Universal Robots PolyScope program: skinkekutterFull.urp

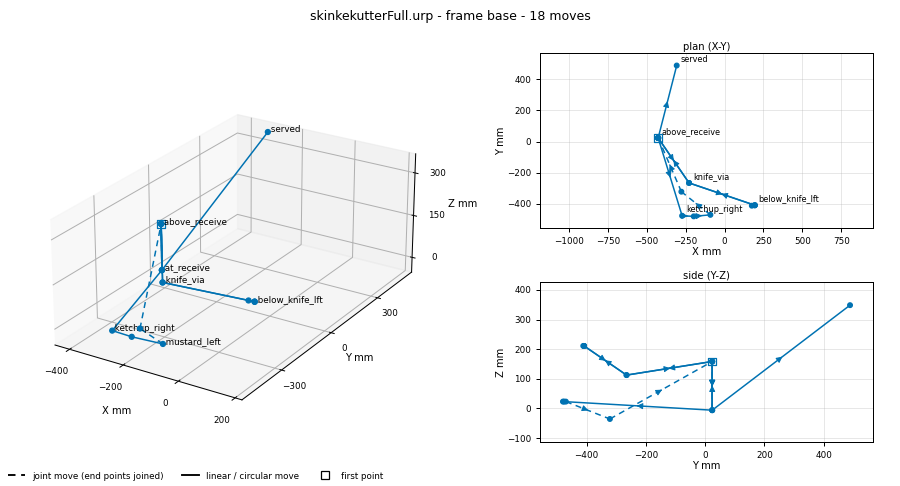
[picture p0: tool path of skinkekutterFull.urp in frame base, 18 of 18 moves have a stored position in this frame; points joined in program order, loops and branches not executed]
Program skinkekutter2 (installation=skinkekutter2 directory=/programs createdIn=0.0.0 lastSavedIn=5.13.0 robotSerialNumber=20185300015)
Calibrated DH parameters: a=[-0.000086, -0.242565, -0.211836, 0.000046, -0.000137, 0]; d=[0.151986, 5.97615, 11.782146, -17.627443, 0.08527, 0.092315]; alpha=[1.571049, 0.003818, 0.001446, 1.57052, -1.5709, 0]; deltaTheta=[0, 0.093783, 0.026843, -0.120628, 0.00001, 0]
Robot Program (runOnlyOnce=true)
  Folder Position bread tray
    MoveL speed 100 mm/s, acceleration 100 mm/s^2 (useActiveTCP=true) feature=Base
      Waypoint above_receive: TCP in base x=-426.247 y=23.581 z=158.427 mm, rx=0.0298 ry=0.0541 rz=-1.4798 rad; joints [-27.463, -23.346, 82.065, -151.039, 88.023, 32.665] deg; TCP offset x=50 y=0 z=0 mm, rx=0 ry=0 rz=0 rad
      Waypoint at_receive: TCP in base x=-426.262 y=23.57 z=-5.894 mm, rx=0.0299 ry=0.0541 rz=-1.4798 rad; joints [-27.518, 14.507, 47.901, -154.728, 88.008, 32.577] deg
  Call wait_for_robot1
  Folder Cut bread
    MoveL speed 100 mm/s, acceleration 100 mm/s^2 (useActiveTCP=true) feature=Base
      Waypoint above_receive: TCP in base x=-426.247 y=23.581 z=158.427 mm, rx=0.0298 ry=0.0541 rz=-1.4798 rad; joints [-27.463, -23.346, 82.065, -151.039, 88.023, 32.665] deg
      Waypoint knife_via: TCP in base x=-227.909 y=-265.427 z=112.534 mm, rx=0.029 ry=0.0408 rz=-1.4657 rad; joints [17.782, -19.961, 117.176, -186.969, 87.596, -11.824] deg
      Waypoint below_knife_lft: TCP in base x=194.493 y=-408.711 z=210.838 mm, rx=-0.0369 ry=-0.025 rz=-1.4267 rad; joints [98.682, -36.96, 96.863, -152.155, 89.61, -90.412] deg
    Force Frame feature=Base; selection=[0, 0, 1, 0, 0, 0]; wrench=[0, 0, 15, 0, 0, 0]; limitsForce=[0.15, 0.15, 0.02, 1.047198, 1.047198, 1.047198]; limitsMotion=[0.1, 0.1, 0.1, 0.349066, 0.349066, 0.349066]
      Loop Counting (count=4) loopVariable(name=Loop_1)
        MoveL speed 50 mm/s, acceleration 100 mm/s^2 (useActiveTCP=true) feature=Base
          Waypoint below_knife_rgt: TCP in base x=175.139 y=-411.516 z=211.031 mm, rx=-0.0369 ry=-0.0249 rz=-1.4266 rad; joints [95.763, -37.722, 98.955, -153.511, 89.721, -87.49] deg
          Waypoint below_knife_lft: TCP in base x=194.493 y=-408.711 z=210.838 mm, rx=-0.0369 ry=-0.025 rz=-1.4267 rad; joints [98.682, -36.96, 96.863, -152.155, 89.61, -90.412] deg
    MoveL speed 100 mm/s, acceleration 100 mm/s^2 (useActiveTCP=true) feature=Base
      Waypoint below_knife_lft: TCP in base x=194.493 y=-408.711 z=210.838 mm, rx=-0.0369 ry=-0.025 rz=-1.4267 rad; joints [98.682, -36.96, 96.863, -152.155, 89.61, -90.412] deg
      Waypoint knife_via: TCP in base x=-227.909 y=-265.427 z=112.534 mm, rx=0.029 ry=0.0408 rz=-1.4657 rad; joints [17.782, -19.961, 117.176, -186.969, 87.596, -11.824] deg
      Waypoint above_receive: TCP in base x=-426.247 y=23.581 z=158.427 mm, rx=0.0298 ry=0.0541 rz=-1.4798 rad; joints [-27.463, -23.346, 82.065, -151.039, 88.023, 32.665] deg
      Waypoint at_receive: TCP in base x=-426.262 y=23.57 z=-5.894 mm, rx=0.0299 ry=0.0541 rz=-1.4798 rad; joints [-27.518, 14.507, 47.901, -154.728, 88.008, 32.577] deg
  Call wait_for_robot1
  Folder To ketchup
    MoveL speed 100 mm/s, acceleration 100 mm/s^2 (useActiveTCP=true) feature=Base
      Waypoint ketchup_right: TCP in base x=-272.485 y=-476.495 z=23.095 mm, rx=0.0562 ry=0.0956 rz=-1.4386 rad; joints [40.987, 22.134, 12.06, -121.923, 84.91, -33.759] deg
  Call wait_for_robot1
  Folder Get ketchup
    MoveL speed 20 mm/s, acceleration 100 mm/s^2 (useActiveTCP=true) feature=Base
      Waypoint ketchup_left: TCP in base x=-198.014 y=-480.033 z=23.107 mm, rx=0.0562 ry=0.0956 rz=-1.4387 rad; joints [47.712, 9.13, 44.649, -140.898, 85.206, -40.474] deg
  Call wait_for_robot1
  Folder Get ketchup
    MoveL speed 20 mm/s, acceleration 100 mm/s^2 (useActiveTCP=true) feature=Base
      Waypoint mustard_left: TCP in base x=-90.886 y=-470.288 z=23.098 mm, rx=0.0562 ry=0.0956 rz=-1.4386 rad; joints [58.449, 2.319, 67.026, -155.571, 85.813, -51.204] deg
  Call wait_for_robot1
  Folder Folder
    MoveJ speed 60 deg/s, acceleration 80 deg/s^2 (useActiveTCP=true) feature=Base
      Waypoint via_back: TCP in base x=-277.299 y=-321.672 z=-35.556 mm, rx=0.063 ry=0.0753 rz=-1.8872 rad; joints [25.168, 14.237, 68.046, -169.906, 86.014, -43.619] deg
      Waypoint above_receive: motionParameters(jointSpeed=1.047198 jointAcceleration=1.396263 cartesianSpeed=0.25 cartesianAcceleration=1.2); TCP in base x=-426.247 y=23.581 z=158.427 mm, rx=0.0298 ry=0.0541 rz=-1.4798 rad; joints [-27.463, -23.346, 82.065, -151.039, 88.023, 32.665] deg
      Waypoint at_receive: TCP in base x=-426.262 y=23.57 z=-5.894 mm, rx=0.0299 ry=0.0541 rz=-1.4798 rad; joints [-27.518, 14.507, 47.901, -154.728, 88.008, 32.577] deg
  Call wait_for_robot1
  MoveL speed 100 mm/s, acceleration 100 mm/s^2 (useActiveTCP=true) feature=Base
    Waypoint served: TCP in base x=-307.263 y=488.731 z=348.51 mm, rx=-0.1494 ry=0.047 rz=1.8704 rad; joints [-71.104, -33.737, 37.032, -85.919, 87.984, -91.584] deg
SubProgram -> wait_for_robot1
SubProgram wait_for_robot1 (keepSynchronizedWithDisk=false)
  Folder Robot1 takes over
    Set DigitalOutput pin=digital_out[4]; digitalValue=1
    Wait Sleep waitTime=0.01
    Set DigitalOutput pin=digital_out[4]; digitalValue=0
    Wait DigitalInput pin=digital_in[0]; digitalValue=1
